FUNCTION_BLOCK EmergencyManagementControl (* Basic Function Block Type *)
  (* Standard: 61499-2 *)
  (* Version 0.0, 7/5/2026, Schneider Electric, Template *)
  PACKAGE SE.Nereda;
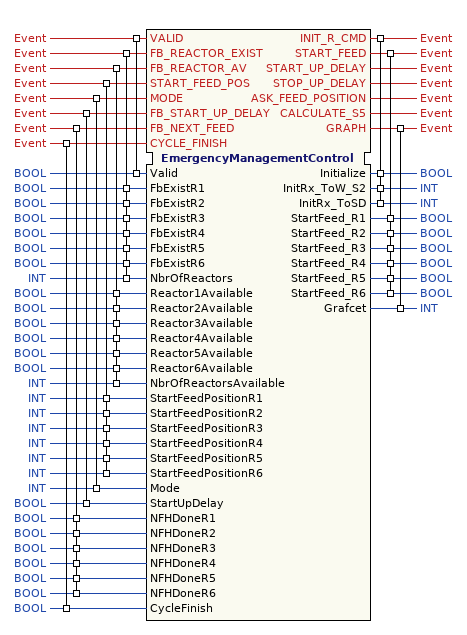
  EVENT_INPUT
    VALID WITH Valid;
    FB_REACTOR_EXIST WITH FbExistR1, FbExistR2, FbExistR3, FbExistR4, FbExistR5, FbExistR6, NbrOfReactors;
    FB_REACTOR_AV WITH Reactor1Available, Reactor2Available, Reactor3Available, Reactor4Available, Reactor5Available, Reactor6Available, NbrOfReactorsAvailable;
    START_FEED_POS WITH StartFeedPositionR1, StartFeedPositionR2, StartFeedPositionR3, StartFeedPositionR4, StartFeedPositionR5, StartFeedPositionR6;
    MODE WITH Mode;
    FB_START_UP_DELAY WITH StartUpDelay;
    FB_NEXT_FEED WITH NFHDoneR6, NFHDoneR1, NFHDoneR2, NFHDoneR3, NFHDoneR4, NFHDoneR5;
    CYCLE_FINISH WITH CycleFinish;
  END_EVENT
  EVENT_OUTPUT
    INIT_R_CMD WITH Initialize, InitRx_ToW_S2, InitRx_ToSD;
    START_FEED WITH StartFeed_R1, StartFeed_R2, StartFeed_R3, StartFeed_R4, StartFeed_R5, StartFeed_R6;
    START_UP_DELAY;
    STOP_UP_DELAY;
    ASK_FEED_POSITION;
    CALCULATE_S5;
    GRAPH WITH Grafcet;
  END_EVENT
  VAR_INPUT
    Valid : BOOL;
    FbExistR1 : BOOL;
    FbExistR2 : BOOL;
    FbExistR3 : BOOL;
    FbExistR4 : BOOL;
    FbExistR5 : BOOL;
    FbExistR6 : BOOL;
    NbrOfReactors : INT;
    Reactor1Available : BOOL;
    Reactor2Available : BOOL;
    Reactor3Available : BOOL;
    Reactor4Available : BOOL;
    Reactor5Available : BOOL;
    Reactor6Available : BOOL;
    NbrOfReactorsAvailable : INT;
    StartFeedPositionR1 : INT;
    StartFeedPositionR2 : INT;
    StartFeedPositionR3 : INT;
    StartFeedPositionR4 : INT;
    StartFeedPositionR5 : INT;
    StartFeedPositionR6 : INT;
    Mode : INT;
    StartUpDelay : BOOL;
    NFHDoneR1 : BOOL;
    NFHDoneR2 : BOOL;
    NFHDoneR3 : BOOL;
    NFHDoneR4 : BOOL;
    NFHDoneR5 : BOOL;
    NFHDoneR6 : BOOL;
    CycleFinish : BOOL;
  END_VAR
  VAR_OUTPUT
    Initialize : BOOL;
    InitRx_ToW_S2 : INT;
    InitRx_ToSD : INT;
    StartFeed_R1 : BOOL;
    StartFeed_R2 : BOOL;
    StartFeed_R3 : BOOL;
    StartFeed_R4 : BOOL;
    StartFeed_R5 : BOOL;
    StartFeed_R6 : BOOL;
    Grafcet : INT;
  END_VAR
  VAR
    InitDone : BOOL;
  END_VAR
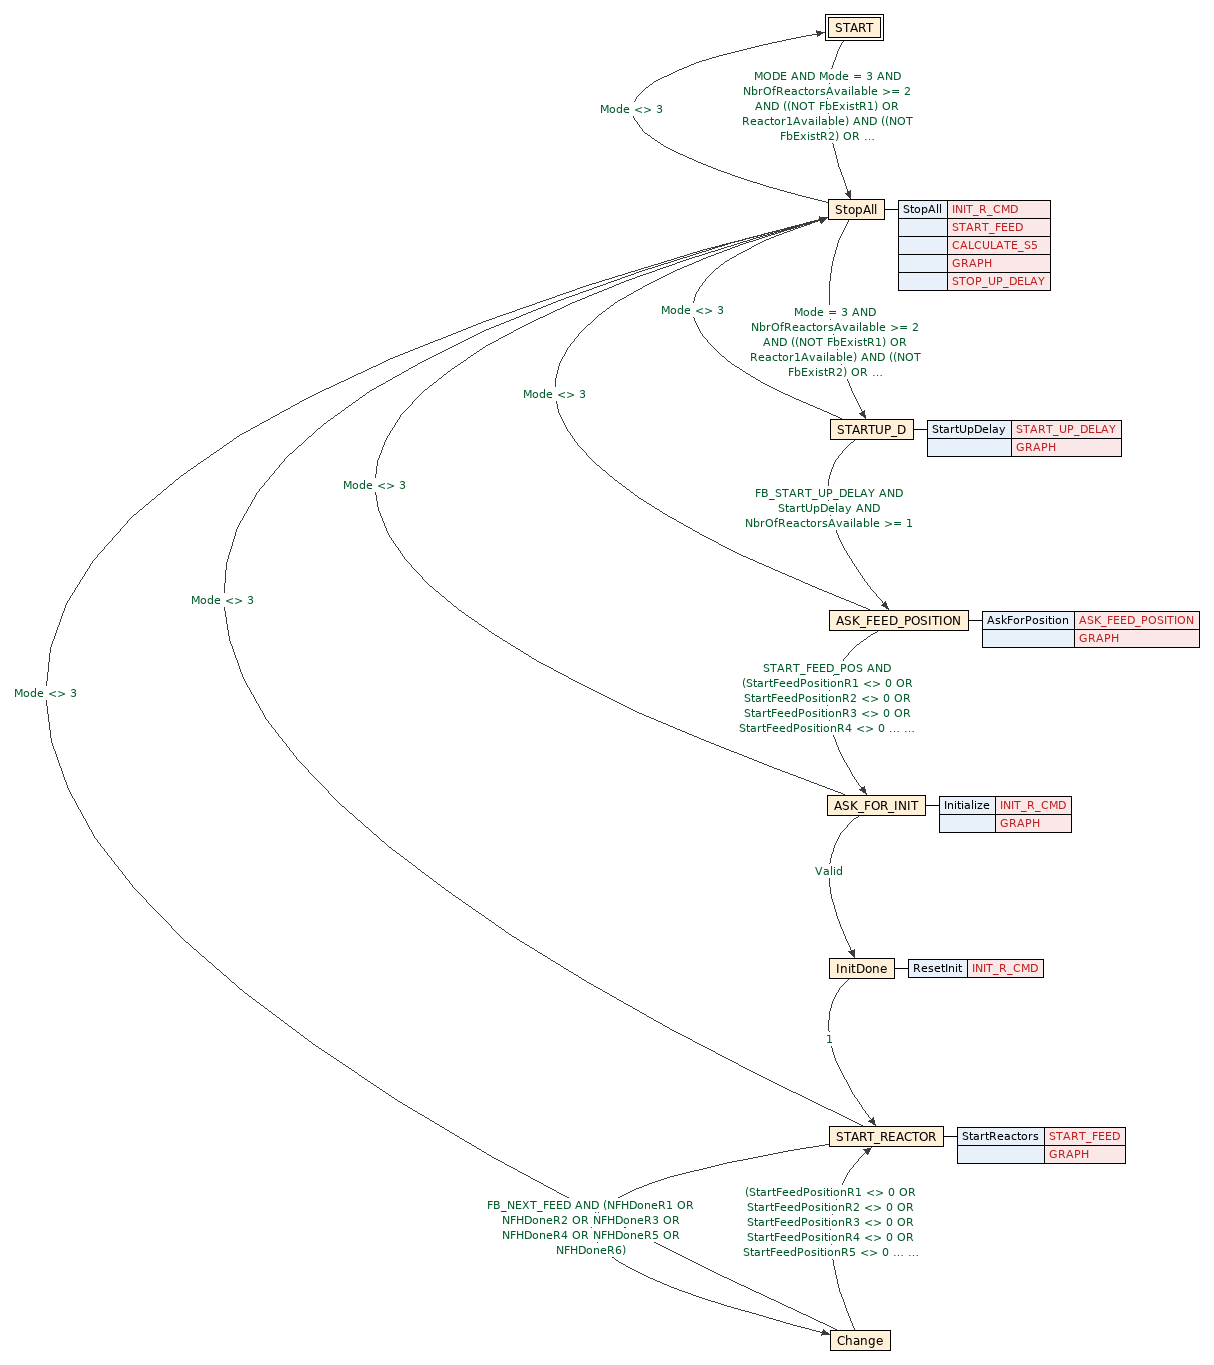
  EC_STATES
    START; (* Initial State *)
    StopAll : StopAll -> INIT_R_CMD, -> START_FEED, -> CALCULATE_S5, -> GRAPH, -> STOP_UP_DELAY;
    ASK_FEED_POSITION : AskForPosition -> ASK_FEED_POSITION, -> GRAPH;
    ASK_FOR_INIT : Initialize -> INIT_R_CMD, -> GRAPH;
    STARTUP_D : StartUpDelay -> START_UP_DELAY, -> GRAPH;
    InitDone : ResetInit -> INIT_R_CMD;
    START_REACTOR : StartReactors -> START_FEED, -> GRAPH;
    Change;
  END_STATES
  EC_TRANSITIONS
    START TO StopAll := MODE AND Mode = 3 AND NbrOfReactorsAvailable >= 2 AND ((NOT FbExistR1) OR Reactor1Available) AND ((NOT FbExistR2) OR Reactor2Available) AND ((NOT FbExistR3) OR Reactor3Available) AND ((NOT FbExistR4) OR Reactor4Available) AND ((NOT FbExistR5) OR Reactor5Available) AND ((NOT FbExistR6) OR Reactor6Available);
    STARTUP_D TO ASK_FEED_POSITION := FB_START_UP_DELAY AND StartUpDelay AND NbrOfReactorsAvailable >= 1;
    StopAll TO START := Mode <> 3;
    ASK_FEED_POSITION TO ASK_FOR_INIT := START_FEED_POS AND (StartFeedPositionR1 <> 0 OR StartFeedPositionR2 <> 0 OR StartFeedPositionR3 <> 0 OR StartFeedPositionR4 <> 0 OR StartFeedPositionR5 <> 0 OR StartFeedPositionR6 <> 0);
    ASK_FOR_INIT TO InitDone := Valid;
    StopAll TO STARTUP_D := Mode = 3 AND NbrOfReactorsAvailable >= 2 AND ((NOT FbExistR1) OR Reactor1Available) AND ((NOT FbExistR2) OR Reactor2Available) AND ((NOT FbExistR3) OR Reactor3Available) AND ((NOT FbExistR4) OR Reactor4Available) AND ((NOT FbExistR5) OR Reactor5Available) AND ((NOT FbExistR6) OR Reactor6Available);
    START_REACTOR TO StopAll := Mode <> 3;
    STARTUP_D TO StopAll := Mode <> 3;
    ASK_FEED_POSITION TO StopAll := Mode <> 3;
    ASK_FOR_INIT TO StopAll := Mode <> 3;
    InitDone TO START_REACTOR := 1;
    START_REACTOR TO Change := FB_NEXT_FEED AND (NFHDoneR1 OR NFHDoneR2 OR NFHDoneR3 OR NFHDoneR4 OR NFHDoneR5 OR NFHDoneR6);
    Change TO START_REACTOR := (StartFeedPositionR1 <> 0 OR StartFeedPositionR2 <> 0 OR StartFeedPositionR3 <> 0 OR StartFeedPositionR4 <> 0 OR StartFeedPositionR5 <> 0 OR StartFeedPositionR6 <> 0);
    Change TO StopAll := Mode <> 3;
  END_TRANSITIONS
  ALGORITHM StopAll IN ST:
;
Grafcet := 10;
InitDone := FALSE;
Initialize := FALSE;
InitRx_ToSD := 0;
InitRx_ToW_S2 := 0;
StartFeed_R1 := FALSE;
StartFeed_R2 := FALSE;
StartFeed_R3 := FALSE;
StartFeed_R4 := FALSE;
StartFeed_R5 := FALSE;
StartFeed_R6 := FALSE;
  END_ALGORITHM
  ALGORITHM Initialize IN ST:
;
Grafcet := 3;
Initialize := TRUE;

//=========================================================
IF FbExistR1 AND StartFeedPositionR1 = 3 THEN
	InitRx_ToSD := 1;
END_IF;

IF FbExistR2 AND StartFeedPositionR2 = 3 THEN
	InitRx_ToSD := 2;
END_IF;

IF FbExistR3 AND StartFeedPositionR3 = 3 THEN
	InitRx_ToSD := 3;
END_IF;

IF FbExistR4 AND StartFeedPositionR4 = 3 THEN
	InitRx_ToSD := 4;
END_IF;

IF FbExistR5 AND StartFeedPositionR5 = 3 THEN
	InitRx_ToSD := 5;
END_IF;

IF FbExistR6 AND StartFeedPositionR6 = 3 THEN
	InitRx_ToSD := 6;
END_IF;

//=========================================================
IF FbExistR1 AND StartFeedPositionR1 = 2 THEN
	InitRx_ToW_S2 := 1;
END_IF;

IF FbExistR2 AND StartFeedPositionR2 = 2 THEN
	InitRx_ToW_S2 := 2;
END_IF;

IF FbExistR3 AND StartFeedPositionR3 = 2 THEN
	InitRx_ToW_S2 := 3;
END_IF;

IF FbExistR4 AND StartFeedPositionR4 = 2 THEN
	InitRx_ToW_S2 := 4;
END_IF;

IF FbExistR5 AND StartFeedPositionR5 = 2 THEN
	InitRx_ToW_S2 := 5;
END_IF;

IF FbExistR6 AND StartFeedPositionR6 = 2 THEN
	InitRx_ToW_S2 := 6;
END_IF;
  END_ALGORITHM
  ALGORITHM StartUpDelay IN ST:
;
Grafcet := 1;
  END_ALGORITHM
  ALGORITHM AskForPosition IN ST:
;
Grafcet := 2;

StartFeed_R1 := FALSE;
StartFeed_R2 := FALSE;
StartFeed_R3 := FALSE;
StartFeed_R4 := FALSE;
StartFeed_R5 := FALSE;
StartFeed_R6 := FALSE;
  END_ALGORITHM
  ALGORITHM ResetInit IN ST:
;
Initialize := FALSE;
InitDone := TRUE;
  END_ALGORITHM
  ALGORITHM StartReactors IN ST:
;
Grafcet := 4;
IF FbExistR1 AND StartFeedPositionR1 = 1 THEN
	StartFeed_R1 := TRUE;

	StartFeed_R2 := FALSE;
	StartFeed_R3 := FALSE;
	StartFeed_R4 := FALSE;
	StartFeed_R5 := FALSE;
	StartFeed_R6 := FALSE;
END_IF;

IF FbExistR2 AND StartFeedPositionR2 = 1 THEN
	StartFeed_R2 := TRUE;

	StartFeed_R1 := FALSE;
	StartFeed_R3 := FALSE;
	StartFeed_R4 := FALSE;
	StartFeed_R5 := FALSE;
	StartFeed_R6 := FALSE;

END_IF;

IF FbExistR3 AND StartFeedPositionR3 = 1 THEN
	StartFeed_R3 := TRUE;

	StartFeed_R1 := FALSE;
	StartFeed_R2 := FALSE;
	StartFeed_R4 := FALSE;
	StartFeed_R5 := FALSE;
	StartFeed_R6 := FALSE;
END_IF;

IF FbExistR4 AND StartFeedPositionR4 = 1 THEN
	StartFeed_R4 := TRUE;

	StartFeed_R1 := FALSE;
	StartFeed_R2 := FALSE;
	StartFeed_R3 := FALSE;
	StartFeed_R5 := FALSE;
	StartFeed_R6 := FALSE;
END_IF;

IF FbExistR5 AND StartFeedPositionR5 = 1 THEN
	StartFeed_R5 := TRUE;

	StartFeed_R1 := FALSE;
	StartFeed_R2 := FALSE;
	StartFeed_R3 := FALSE;
	StartFeed_R4 := FALSE;
	StartFeed_R6 := FALSE;
END_IF;

IF FbExistR6 AND StartFeedPositionR6 = 1 THEN
	StartFeed_R6 := TRUE;

	StartFeed_R1 := FALSE;
	StartFeed_R2 := FALSE;
	StartFeed_R3 := FALSE;
	StartFeed_R4 := FALSE;
	StartFeed_R5 := FALSE;
END_IF;
  END_ALGORITHM
END_FUNCTION_BLOCK
